{attribute 'linkalways'} 
{attribute 'no_explicit_call' := 'This FB is a CLASS and must be accessed using methods or properties'}
{attribute 'enable_dynamic_creation'}
FUNCTION_BLOCK Node_F_VN_AppendToContainer_TcVnVector2_DINT EXTENDS VisionNode
VAR
    aElement : _TcVnVector2_DINT;
    ipContainer : _ITcVnContainer;
    hrPrev : _HRESULT(S_OK);
	hresult : _HRESULT(S_OK);
END_VAR

METHOD PUBLIC  Clone : I_Node
VAR
	pNode : POINTER TO Node_F_VN_AppendToContainer_TcVnVector2_DINT;
END_VAR
pNode := __NEW(Node_F_VN_AppendToContainer_TcVnVector2_DINT);
Clone := pNode^;
END_METHOD

METHOD FB_init : BOOL
VAR_INPUT
	bInitRetains : BOOL; // if TRUE, the retain variables are initialized (warm start / cold start)
	bInCopyCode : BOOL;  // if TRUE, the instance afterwards gets moved into the copy code (online change)
END_VAR
AddInput('aElement', aElement);
AddInput('ipContainer', ipContainer);
AddInput('hrPrev', hrPrev);
AddOutput('ipContainer', ipContainer);
AddOutput('hresult',hresult);
END_METHOD

METHOD PROTECTED OnExecute : HRESULT
hresult.Value := F_VN_AppendToContainer_TcVnVector2_DINT(
    aElement := aElement.Value,
	ipContainer := ipContainer.Value,
	hrPrev:= hrPrev.Value);
END_METHOD

METHOD PUBLIC PreExecutionCheck
VAR_INPUT
	Check : I_PreExecutionChecks;
END_VAR
Check.IsTrue(ipContainer.IsValid, 'ipContainer must be a valid container');
END_METHOD

END_FUNCTION_BLOCK

(* stored: Version 1.1.0.1, ProductVersion 3.1.4024.13
   POU Node_F_VN_AppendToContainer_TcVnVector2_DINT: Id {c5f63b3b-bbbd-4204-b58e-0d5822379fbd}, SpecialFunc None
   Folder Constructor: Id {175e22dc-c2b5-483a-b128-9a8df404d255}
   Method Clone: Id {876d68ef-ff3b-4a45-a2d1-8f3c4b2d6e7c}
   Method FB_init: Id {960a98ae-d545-4064-b836-ad5f01db6406}
   Method OnExecute: Id {d08f1950-d60e-4aa2-a65f-6c7bb796134e}
   Method PreExecutionCheck: Id {4fe949d6-1926-49da-9a11-238a8bf809d9} *)
